{attribute 'linkalways'}
{attribute 'hide_all_locals'}
FUNCTION_BLOCK ValueLintRead EXTENDS ValueBase IMPLEMENTS ValueRead
VAR
	thisValue : LINT;
END_VAR

{attribute 'call_after_global_init_slot' := '1'}
{attribute 'call_after_online_change_slot' := '1'}
METHOD PROTECTED GetThisAnyType
VAR_INPUT
END_VAR
thisAnyType := ToAnyType(thisValue);
END_METHOD

METHOD GetAsType : BOOL
VAR_INPUT
	destination : __SYSTEM.AnyType;
END_VAR
GetAsType := ConvertAnyType(thisAnyType, destination);
END_METHOD

METHOD GetAsString : T_MaxString
VAR_INPUT
END_VAR
GetAsString := TO_STRING(thisValue);
END_METHOD

METHOD Get : BOOL
VAR_INPUT
	destination : ANY;
END_VAR
Get := ConvertAnyType(thisAnyType, destination);
END_METHOD

METHOD FB_init : BOOL
VAR_INPUT
	bInitRetains : BOOL; // if TRUE, the retain variables are initialized (warm start / cold start)
	bInCopyCode : BOOL;  // if TRUE, the instance afterwards gets moved into the copy code (online change)
END_VAR
_ValueType := __SYSTEM.TYPE_CLASS.TYPE_LINT;
END_METHOD

{attribute 'monitoring' := 'call'}
PROPERTY Value : LINT
GET
Value := thisValue;
END_GET
END_PROPERTY

END_FUNCTION_BLOCK

(* stored: Version 1.1.0.1
   POU ValueLintRead: Id {901a3e76-f083-4baa-ae99-6198fcffca44}, SpecialFunc None
   Method GetThisAnyType: Id {48a4293a-4c80-4fbe-a089-26cfbe5c8e7d}
   Method GetAsType: Id {e58d8fcb-72ad-49ff-badb-b984738de588}
   Method GetAsString: Id {3ede59d7-f771-4d19-a692-47eded7895f8}
   Method Get: Id {21b67296-5f07-4f4f-a091-2597d385ab81}
   Method FB_init: Id {3601ec52-76f0-4434-b508-f1d45cea04cc}
   Property Value: Id {d743305d-94d9-4ebc-b75c-2e51f9a9bd0d}
   Get Get: Id {9d5ba8f0-e943-425c-a62e-02cebf46c83c} *)
